FUNCTION_BLOCK FT_PT2_AR (* AR-Adapter-Wrapper um OSCAT FT_PT2 (PT2-Tiefpassfilter 2. Ordnung) - bruckt zwischen adapter und OSCAT, ohne dass eine der beiden Basisbibliotheken von der anderen abhaengt. TM (Zeitkonstante) als ATM-Socket (kein Klartext-InputVar, sauber initialisierbar ueber initval_ATM), D/K als Klartext-InputVars durchgereicht *)
  (* Standard: 61499-2; Description: Copyright (c) 2026 Meisterschulen am Ostbahnhof This program and the accompanying materials are made available under the terms of the Eclipse Public License 2.0 which is available at https://www.eclipse.org/legal/epl-2.0/ SPDX-License-Identifier: EPL-2.0 *)
  (* Version 1.0, 2026-09-17, Franz Höpfinger, Meisterschulen am Ostbahnhof, Initial implementation of FT_PT2_AR wrapper FB (Franz: 'portiere diese Bausteine hier her', OSCAT_basic FT_PT2.TcPOU) - E_D_FF_ANY als Aenderungsfilter (EO/AR_OUT.E1 nur bei tatsaechlicher Wertaenderung), analog ROUND_AR/FT_DERIV_AR/FT_PT1_AR in diesem Projekt. TM als ATM-Socket statt Klartext-InputVar (Section 13 des iec61499-creator-Skills), D/K als Klartext-InputVars (statisch pro Aufruf, wie K/run bei FT_DERIV_AR). FT_PT2.fbt selbst existierte bereits im Projekt (Version 1.5, 2025-12-21) - hier nur der fehlende Adapter-Wrapper ergaenzt. *)
  PACKAGE OSCAT_adapter::Control;
  (* Documentation:
  FT_PT2_AR
   🇩🇪 Deutsch
   AR-Adapter-Wrapper um OSCAT::Basic::POUs::Engineering::Control::FT_PT2 (Filter 2. Ordnung mit programmierbarer Zeitkonstante TM, Daempfung D und Faktor K). TM ist ein ATM-Socket (kein Klartext-InputVar) - an der Instanziierungsstelle ueber adapter::types::unidirectional::TIME::initval::initval_ATM zu initialisieren (Section 13 des iec61499-creator-Skills). D/K bleiben Klartext-InputVars, da rein statisch pro Aufruf und ueber Parameter setzbar wie bei FT_DERIV_AR.
   Reine Adapter-Grenze
    - AR_IN (Socket, AR): Eingangssignal (REAL)
   - TM (Socket, ATM): Zeitkonstante
   - AR_OUT (Plug, AR): gefilterter Ausgangswert (REAL)
    E_D_FF_ANY filtert Aenderungen: AR_OUT.E1 feuert nur, wenn sich der gefilterte Wert seit dem letzten Aufruf tatsaechlich geaendert hat - gleiches Muster wie bei ROUND_AR/FT_DERIV_AR/FT_PT1_AR in diesem Projekt.
   INIT/INITO/RST werden 1:1 an FT_PT2.EINIT/.INITO/.RST durchgereicht. Bleibt INIT unverdrahtet, feuert es einmalig beim Deployment automatisch (Standardkonvention fuer unverdrahtete EInit-Events).
   Warum ein eigener Wrapper?
   FT_PT2 ist ein reines OSCAT-FB (SimpleFB, zustandsbehaftet, kapselt intern zwei INTEGRATE-Instanzen) ohne Adapter-Schnittstelle. adapter soll nicht von OSCAT abhaengen (und umgekehrt) - die Bruecke liegt daher in diesem dritten Bibliotheksprojekt (OSCAT_adapter), das von beiden abhaengt.
   🇬🇧 English
   AR-adapter wrapper around OSCAT::Basic::POUs::Engineering::Control::FT_PT2 (2nd-order filter with programmable time constant TM, damping D and factor K). TM is an ATM socket (not a plain InputVar) - initialize it at the instantiation site via adapter::types::unidirectional::TIME::initval::initval_ATM (per section 13 of the iec61499-creator skill). D/K stay plain InputVars, since they're purely static per call and settable via Parameter, like on FT_DERIV_AR.
   Pure adapter boundary
    - AR_IN (socket, AR): input signal (REAL)
   - TM (socket, ATM): time constant
   - AR_OUT (plug, AR): filtered output value (REAL)
    E_D_FF_ANY filters changes: AR_OUT.E1 only fires when the filtered value actually changed since the last call - same pattern as ROUND_AR/FT_DERIV_AR/FT_PT1_AR in this project.
   INIT/INITO/RST are passed through 1:1 to FT_PT2.EINIT/.INITO/.RST. If INIT is left unconnected, it auto-fires once at deployment (standard convention for unconnected EInit events).
   Why a dedicated wrapper?
   FT_PT2 is a plain OSCAT FB (SimpleFB, stateful, internally wraps two INTEGRATE instances) with no adapter interface. adapter must not depend on OSCAT (nor vice versa) - the bridge lives in this third library project (OSCAT_adapter), which depends on both.
  *)
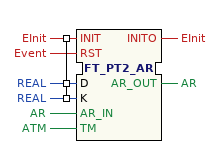
  EVENT_INPUT
    INIT : EInit WITH D, K; (* Service Initialization (durchgereicht an FT_PT2.EINIT) *)
    RST; (* Filter zuruecksetzen (durchgereicht an FT_PT2.RST) *)
  END_EVENT
  EVENT_OUTPUT
    INITO : EInit; (* Initialization Confirm *)
  END_EVENT
  VAR_INPUT
    D : REAL; (* Daempfungsfaktor (durchgereicht an FT_PT2.D) *)
    K : REAL := 1.0; (* Faktor (durchgereicht an FT_PT2.K) *)
  END_VAR
  SOCKETS
    AR_IN : adapter::types::unidirectional::AR; (* Eingangssignal (REAL) *)
    TM : adapter::types::unidirectional::ATM; (* Zeitkonstante (durchgereicht an FT_PT2.TM) *)
  END_SOCKETS
  PLUGS
    AR_OUT : adapter::types::unidirectional::AR; (* Gefilterter Ausgangswert (REAL, durchgereicht von FT_PT2.out) *)
  END_PLUGS
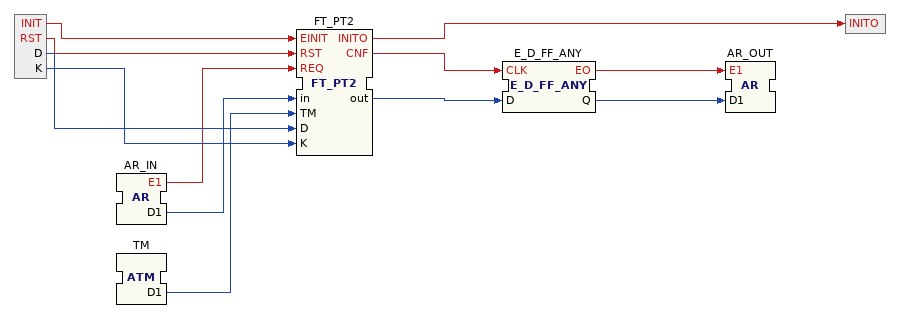
  FBS
    FT_PT2 : OSCAT::Basic::POUs::Engineering::Control::FT_PT2;
    E_D_FF_ANY : iec61499::events::E_D_FF_ANY;
  END_FBS
  EVENT_CONNECTIONS
    INIT TO FT_PT2.EINIT;
    FT_PT2.INITO TO INITO;
    RST TO FT_PT2.RST;
    AR_IN.E1 TO FT_PT2.REQ;
    FT_PT2.CNF TO E_D_FF_ANY.CLK;
    E_D_FF_ANY.EO TO AR_OUT.E1;
  END_CONNECTIONS
  DATA_CONNECTIONS
    AR_IN.D1 TO FT_PT2.in;
    TM.D1 TO FT_PT2.TM;
    D TO FT_PT2.D;
    K TO FT_PT2.K;
    FT_PT2.out TO E_D_FF_ANY.D;
    E_D_FF_ANY.Q TO AR_OUT.D1;
  END_CONNECTIONS
END_FUNCTION_BLOCK
